{attribute addProperty BoxType "EKM1101-0000-0016"}
{attribute addProperty Id "StatusAT %I*Status_F0C7FE3C3241ValueAT %I*REAL32417"}
{attribute addProperty CRC "3207848129"}
{attribute addProperty SizeInBites "64"}
{attribute addProperty SizeInBytes "8"}
TYPE MMS_Voltage_Us_In_Inputs_BF33E0C1 :
STRUCT
	{attribute addProperty Name "Status"}
	Status AT %I* : Status_F0C7FE3C;
	{attribute addProperty Name "Value"}
	Value AT %I* : REAL;
END_STRUCT
END_TYPE

(* stored: Version 1.2.0.0, ProductVersion 3.1.4024.9
   DUT MMS_Voltage_Us_In_Inputs_BF33E0C1: Id {f91ebfcd-011d-4f15-9033-dc8995eae34d} *)
